KUKA KRL program: kuka_eki_command_server_dep.sub, kuka_eki_command_server_dep.dat

--- kuka_eki_command_server_dep.sub ---
&ACCESS RVP
&PARAM EDITMASK = *
&PARAM TEMPLATE = C:\KRC\Roboter\Template\submit
def kuka_eki_command_server()
   ;FOLD DECLARATIONS
   ;FOLD USER DECL
   ; local vairable declarations
   decl int elements_read
   decl real laser_temp

   eki_hw_iface_init() ; socket connection

   laser_temp = 0

   parameters[1] = $POS_ACT.X
   parameters[2] = $POS_ACT.Y
   parameters[3] = $POS_ACT.Z
   parameters[4] = $POS_ACT.A
   parameters[5] = $POS_ACT.B
   parameters[6] = $POS_ACT.C

   cartesian_target.X = $POS_ACT.X
   cartesian_target.Y = $POS_ACT.Y
   cartesian_target.Z = $POS_ACT.Z
   cartesian_target.A = $POS_ACT.A
   cartesian_target.B = $POS_ACT.B
   cartesian_target.C = $POS_ACT.C

   instruction_code = 0


   loop
      elements_read = eki_get_temperature(laser_temp) ; checking the laser temp with Arduino reading
      if laser_temp>26 then
      $OUT[3]=FALSE
      $OUT[1]=FALSE
      endif

      elements_read = eki_hw_iface_get()  ; Get new command from buffer


      SWITCH (instruction_code)
      CASE 1
         ; cartesian motion command, phrase parameters into global variable cartesian_target
         cartesian_target.X = parameters[1]
         cartesian_target.Y = parameters[2]
         cartesian_target.Z = parameters[3]
         cartesian_target.A = parameters[4]
         cartesian_target.B = parameters[5]
         cartesian_target.C = parameters[6]
         MsgNotify("Cartesian target command received and set",,,,)

      DEFAULT
         cartesian_target.X = $POS_ACT.X
         cartesian_target.Y = $POS_ACT.Y
         cartesian_target.Z = $POS_ACT.Z
         cartesian_target.A = $POS_ACT.A
         cartesian_target.B = $POS_ACT.B
         cartesian_target.C = $POS_ACT.C
      ENDSWITCH
   endloop


end



def eki_hw_iface_init()
   decl eki_status eki_ret

   ; Setup interrupts
   ; Interrupt 15 - Connection cleanup on client disconnect
   global interrupt decl 15 when $flag[1]==false do eki_hw_iface_reset()
   interrupt on 15
   ; Interrupt 16 - Timer interrupt for periodic state transmission
   global interrupt decl 16 when $timer_flag[1]==true do eki_hw_iface_send()
   interrupt on 16
   wait sec 0.012          ; Wait for next interpolation cycle
   $timer[1] = -200        ; Time in [ms] before first interrupt call
   $timer_stop[1] = false  ; Start timer 1

   ; Create and open EKI interface
   eki_ret = eki_init("EkiCommandServer")
   eki_ret = eki_open("EkiCommandServer")
   MsgNotify("ROS connection established",,,,)
end



def eki_hw_iface_send()
   decl eki_status eki_ret
   decl real vel_percent

   if $flag[1] then  ; If connection alive
      ; Load state values into xml structure
      ; position
      eki_ret = eki_setreal("EkiCommandServer", "RobotState/Pos/@A1", $axis_act_meas.a1)
      eki_ret = eki_setreal("EkiCommandServer", "RobotState/Pos/@A2", $axis_act_meas.a2)
      eki_ret = eki_setreal("EkiCommandServer", "RobotState/Pos/@A3", $axis_act_meas.a3)
      eki_ret = eki_setreal("EkiCommandServer", "RobotState/Pos/@A4", $axis_act_meas.a4)
      eki_ret = eki_setreal("EkiCommandServer", "RobotState/Pos/@A5", $axis_act_meas.a5)
      eki_ret = eki_setreal("EkiCommandServer", "RobotState/Pos/@A6", $axis_act_meas.a6)
      ; velocity
      ;eki_ret = eki_setreal("EkiCommandServer", "RobotState/Vel/@A1", $vel_axis_act[1] * $vel_axis_ma[1] / 100.0)
      ;eki_ret = eki_setreal("EkiCommandServer", "RobotState/Vel/@A2", $vel_axis_act[2] * $vel_axis_ma[2] / 100.0)
      ;eki_ret = eki_setreal("EkiCommandServer", "RobotState/Vel/@A3", $vel_axis_act[3] * $vel_axis_ma[3] / 100.0)
      ;eki_ret = eki_setreal("EkiCommandServer", "RobotState/Vel/@A4", $vel_axis_act[4] * $vel_axis_ma[4] / 100.0)
      ;eki_ret = eki_setreal("EkiCommandServer", "RobotState/Vel/@A5", $vel_axis_act[5] * $vel_axis_ma[5] / 100.0)
      ;eki_ret = eki_setreal("EkiCommandServer", "RobotState/Vel/@A6", $vel_axis_act[6] * $vel_axis_ma[6] / 100.0)
      ; effort
      ;eki_ret = eki_setreal("EkiCommandServer", "RobotState/Eff/@A1", $torque_axis_act[1])
      ;eki_ret = eki_setreal("EkiCommandServer", "RobotState/Eff/@A2", $torque_axis_act[2])
      ;eki_ret = eki_setreal("EkiCommandServer", "RobotState/Eff/@A3", $torque_axis_act[3])
      ;eki_ret = eki_setreal("EkiCommandServer", "RobotState/Eff/@A4", $torque_axis_act[4])
      ;eki_ret = eki_setreal("EkiCommandServer", "RobotState/Eff/@A5", $torque_axis_act[5])
      ;eki_ret = eki_setreal("EkiCommandServer", "RobotState/Eff/@A6", $torque_axis_act[6])
      ; interface state
      eki_ret = eki_checkbuffer("EkiCommandServer", "CommandServer/@InstructionCode")
      eki_ret = eki_setint("EkiCommandServer", "RobotState/CommandServer/@Size", eki_ret.buff)

      ; Send xml structure
      if $flag[1] then  ; Make sure connection hasn't died while updating xml structure
         eki_ret = eki_send("EkiCommandServer", "RobotState")
      endif
   endif

   ; Set timer for next interrupt [ms]
   $timer[1] = -10  ; ~10 ms for above send + 10 ms interrupt timer -> ~50 Hz state transmission
end



deffct int eki_hw_iface_available()
   decl eki_status eki_ret

   if not $flag[1] then
      return 0
   endif

   eki_ret = eki_checkbuffer("EkiCommandServer", "CommandServer/@InstructionCode")
   return eki_ret.buff
endfct


; eki_hw_iface_get: phrase command
; Tries to read most recent message from buffer. q left unchanged if empty.
; Returns number of elements read.
deffct int eki_hw_iface_get()
   decl eki_status eki_ret

   if not $flag[1] then
      return 0
   endif

   eki_ret = eki_checkbuffer("EkiCommandServer", "CommandServer/@InstructionCode")
   if eki_ret.buff <= 0 then
     return 0
   endif

   eki_ret = eki_getint("EkiCommandServer", "CommandServer/@InstructionCode", instruction_code)
   eki_ret = eki_getreal("EkiCommandServer", "CommandServer/Parameters/@P1", parameters[1])
   eki_ret = eki_getreal("EkiCommandServer", "CommandServer/Parameters/@P2", parameters[2])
   eki_ret = eki_getreal("EkiCommandServer", "CommandServer/Parameters/@P3", parameters[3])
   eki_ret = eki_getreal("EkiCommandServer", "CommandServer/Parameters/@P4", parameters[4])
   eki_ret = eki_getreal("EkiCommandServer", "CommandServer/Parameters/@P5", parameters[5])
   eki_ret = eki_getreal("EkiCommandServer", "CommandServer/Parameters/@P6", parameters[6])

   ; length = StrLen(instruction_code)
   ; success = StrToREAL(CHAR receive_string[256], REAL instruction_code)

   return 1
endfct



deffct int eki_get_temperature(temp :out)
   decl eki_status eki_ret
   decl real temp

   if not $flag[1] then
      return 0
   endif

   eki_ret = eki_checkbuffer("EkiCommandServer", "CommandServer/Temp/@Laser")
   if eki_ret.buff <= 0 then
     return 0
   endif

   eki_ret = eki_getreal("EkiCommandServer", "CommandServer/Temp/@Laser", temp)
   return 1
endfct


def eki_hw_iface_reset()
   decl eki_status eki_ret

   eki_ret = eki_clear("EkiCommandServer")
   eki_ret = eki_init("EkiCommandServer")
   eki_ret = eki_open("EkiCommandServer")
end

--- kuka_eki_command_server_dep.dat ---
&ACCESS RVO
&PARAM EDITMASK = *
&PARAM TEMPLATE = C:\KRC\Roboter\Template\submit
defdat kuka_eki_command_server public
;FOLD EXTERNAL DECLARATIONS;%{PE}%MKUKATPBASIS,%CEXT,%VCOMMON,%P
;FOLD BASISTECH EXT;%{PE}%MKUKATPBASIS,%CEXT,%VEXT,%P
EXT  BAS (BAS_COMMAND  :IN,REAL  :IN )
DECL INT SUCCESS
;ENDFOLD (BASISTECH EXT)
;FOLD USER EXT;%{E}%MKUKATPUSER,%CEXT,%VEXT,%P
;Make your modifications here

;ENDFOLD (USER EXT)
;ENDFOLD (EXTERNAL DECLARATIONS)
decl global INT instruction_code      ; identify which command (i.e, velocity, motion, laser, etc)
decl global real parameters[6]        ; number of received parameters in real value
decl global frame cartesian_target    ; frame is a sturct, X, Y, Z, A, B, C
;decl global pos cartesian_target_pos  ;pos: X, Y, Z, A, B, C, INT S, T
enddat
